PROGRAM BancoDeDados
VAR_INPUT
	InsertMarcha: InsertBD_Comandos;
	InsertParada: InsertBD_Comandos;
	ComandoSalvar:ARRAY[1..200] OF BOOL;
	bExecuteInsert		: BOOL; 
END_VAR
VAR
	Parte1Comandos	:STRING[100];
	Parte2Comandos	:STRING;
	Parte3Comandos	:STRING;
	RecordInsert	:FB_DBRecordInsert_EX;
	sCmdInsert		:T_MaxString;
	bInsertBusy		:BOOL;
	bInsertError	:BOOL;
	bInsertErrID	:UDINT;
	nRecords		:UDINT;
	
	Teste: BOOL;
END_VAR



//Código de erro 1142 - Usuário sem permissão para fazer o insert
//Código de erro 1146 - Tabela não encontrada
//Código de erro 1064 - Erro de sintaxe

//Pedaços do comando SQL para ficar melhor a montagem no uso delas
Parte1Comandos := 'INSERT INTO `comandos` (`comando`, `data_hora`, `usuario`, `serial_maquina`) VALUES (';
Parte2Comandos := CONCAT(', CURRENT_TIMESTAMP,$'', Main.NomeUsuario);
Parte3Comandos := CONCAT('$', $'', CONCAT(Main.SerialDaMaquina, '$')'));

RecordInsert(
	sNetID:= '127.0.0.1.1.1', //String containing the AMS network ID of the target device, at which the ADS command is directed.
	hDBID:= 1, // Indicates the ID of the database to be used.
	pCmdAddr:= ADR(sCmdInsert), //Pointer to the executing INSERT command
	cbCmdSize:= SIZEOF(sCmdInsert), //Indicates the length of the INSERT command.
	bExecute:= bExecuteInsert, 
	tTimeout:= T#5S, 
	bBusy=> bInsertBusy, 
	bError=> bInsertError, 
	nErrID=> bInsertErrID);
	

//----------------------- Comandos de funcionamento da máquina -----------------------//
{region "Comandos da máquina"}
//Marcha
bExecuteInsert := FALSE;
IF ComandoSalvar[1] THEN
	InsertMarcha(Insert:= TRUE, NomeComando:= 'MARCHA', InsertOut=> bExecuteInsert, Comando=> sCmdInsert);
	ComandoSalvar[1] := FALSE;
END_IF

//Parar
IF ComandoSalvar[2] THEN
	InsertParada(Insert:= TRUE, NomeComando:= 'PARADA', InsertOut=> bExecuteInsert, Comando=> sCmdInsert);
	ComandoSalvar[2] := FALSE;
END_IF

//Manual
IF ComandoSalvar[3] THEN
	InsertParada(Insert:= TRUE, NomeComando:= 'MAQ. EM MANUAL', InsertOut=> bExecuteInsert, Comando=> sCmdInsert);
	ComandoSalvar[3] := FALSE;
END_IF

//Auto
IF ComandoSalvar[4] THEN
	InsertParada(Insert:= TRUE, NomeComando:= 'MAQ. EM AUTOM.', InsertOut=> bExecuteInsert, Comando=> sCmdInsert);
	ComandoSalvar[4] := FALSE;
END_IF

//Fechar Ordem
IF ComandoSalvar[5] THEN
	InsertParada(Insert:= TRUE, NomeComando:= 'FECHAR ORDEM', InsertOut=> bExecuteInsert, Comando=> sCmdInsert);
	ComandoSalvar[5] := FALSE;
END_IF

//Aceitar lote
IF ComandoSalvar[6] THEN
	InsertParada(Insert:= TRUE, NomeComando:= 'ACEITAR LOTE', InsertOut=> bExecuteInsert, Comando=> sCmdInsert);
	ComandoSalvar[6] := FALSE;
END_IF

//Uma batelada
IF ComandoSalvar[7] THEN
	InsertParada(Insert:= TRUE, NomeComando:= 'UMA BATELADA', InsertOut=> bExecuteInsert, Comando=> sCmdInsert);
	ComandoSalvar[7] := FALSE;
END_IF

//Contínuo
IF ComandoSalvar[8] THEN
	InsertParada(Insert:= TRUE, NomeComando:= 'CONTÍNUO', InsertOut=> bExecuteInsert, Comando=> sCmdInsert);
	ComandoSalvar[8] := FALSE;
END_IF

//Pausa
IF ComandoSalvar[9] THEN
	InsertParada(Insert:= TRUE, NomeComando:= 'PAUSA', InsertOut=> bExecuteInsert, Comando=> sCmdInsert);
	ComandoSalvar[9] := FALSE;
END_IF
{endregion}


//----------------------- Acionamento manual das válvulas -----------------------//
{region "Válvulas Circuito 1"}
//------------------- Válvulas Circuito 1 -------------------//

//Circuito 1 Valvula 1 manual
IF ComandoSalvar[10] THEN
	InsertParada(Insert:= TRUE, NomeComando:= 'VALV. 1 CIRC. 1 MANUAL', InsertOut=> bExecuteInsert, Comando=> sCmdInsert);
	ComandoSalvar[10] := FALSE;
END_IF

//Circuito 1 Valvula 2 manual
IF ComandoSalvar[11] THEN
	InsertParada(Insert:= TRUE, NomeComando:= 'VALV. 2 CIRC. 1 MANUAL', InsertOut=> bExecuteInsert, Comando=> sCmdInsert);
	ComandoSalvar[11] := FALSE;
END_IF

//Circuito 1 Valvula 3 manual
IF ComandoSalvar[12] THEN
	InsertParada(Insert:= TRUE, NomeComando:= 'VALV. 3 CIRC. 1 MANUAL', InsertOut=> bExecuteInsert, Comando=> sCmdInsert);
	ComandoSalvar[12] := FALSE;
END_IF

//Circuito 1 Valvula 4 manual
IF ComandoSalvar[13] THEN
	InsertParada(Insert:= TRUE, NomeComando:= 'VALV. 4 CIRC. 1 MANUAL', InsertOut=> bExecuteInsert, Comando=> sCmdInsert);
	ComandoSalvar[13] := FALSE;
END_IF	  
{endregion}

{region "Válvulas Circuito 2"}
//------------------- Válvulas Circuito 2 -------------------//

//Circuito 2 Valvula 1 manual
IF ComandoSalvar[14] THEN
	InsertParada(Insert:= TRUE, NomeComando:= 'VALV. 1 CIRC. 2 MANUAL', InsertOut=> bExecuteInsert, Comando=> sCmdInsert);
	ComandoSalvar[14] := FALSE;
END_IF

//Circuito 2 Valvula 2 manual
IF ComandoSalvar[15] THEN
	InsertParada(Insert:= TRUE, NomeComando:= 'VALV. 2 CIRC. 2 MANUAL', InsertOut=> bExecuteInsert, Comando=> sCmdInsert);
	ComandoSalvar[15] := FALSE;
END_IF

//Circuito 2 Valvula 3 manual
IF ComandoSalvar[16] THEN
	InsertParada(Insert:= TRUE, NomeComando:= 'VALV. 3 CIRC. 2 MANUAL', InsertOut=> bExecuteInsert, Comando=> sCmdInsert);
	ComandoSalvar[16] := FALSE;
END_IF

//Circuito 2 Valvula 4 manual
IF ComandoSalvar[17] THEN
	InsertParada(Insert:= TRUE, NomeComando:= 'VALV. 4 CIRC. 2 MANUAL', InsertOut=> bExecuteInsert, Comando=> sCmdInsert);
	ComandoSalvar[17] := FALSE;
END_IF
{endregion}

{region "Válvulas Circuito 3"}
//------------------- Válvulas Circuito 3 -------------------//

//Circuito 3 Valvula 1 manual
IF ComandoSalvar[18] THEN
	InsertParada(Insert:= TRUE, NomeComando:= 'VALV. 1 CIRC. 3 MANUAL', InsertOut=> bExecuteInsert, Comando=> sCmdInsert);
	ComandoSalvar[18] := FALSE;
END_IF

//Circuito 3 Valvula 2 manual
IF ComandoSalvar[19] THEN
	InsertParada(Insert:= TRUE, NomeComando:= 'VALV. 2 CIRC. 3 MANUAL', InsertOut=> bExecuteInsert, Comando=> sCmdInsert);
	ComandoSalvar[19] := FALSE;
END_IF

//Circuito 3 Valvula 3 manual
IF ComandoSalvar[20] THEN
	InsertParada(Insert:= TRUE, NomeComando:= 'VALV. 3 CIRC. 3 MANUAL', InsertOut=> bExecuteInsert, Comando=> sCmdInsert);
	ComandoSalvar[20] := FALSE;
END_IF

//Circuito 3 Valvula 4 manual
IF ComandoSalvar[21] THEN
	InsertParada(Insert:= TRUE, NomeComando:= 'VALV. 4 CIRC. 3 MANUAL', InsertOut=> bExecuteInsert, Comando=> sCmdInsert);
	ComandoSalvar[21] := FALSE;
END_IF
{endregion}

{region "Válvulas Circuito 4"}
//------------------- Válvulas Circuito 4 -------------------//

//Circuito 4 Valvula 1 manual
IF ComandoSalvar[22] THEN
	InsertParada(Insert:= TRUE, NomeComando:= 'VALV. 1 CIRC. 4 MANUAL', InsertOut=> bExecuteInsert, Comando=> sCmdInsert);
	ComandoSalvar[22] := FALSE;
END_IF

//Circuito 4 Valvula 2 manual
IF ComandoSalvar[23] THEN
	InsertParada(Insert:= TRUE, NomeComando:= 'VALV. 2 CIRC. 4 MANUAL', InsertOut=> bExecuteInsert, Comando=> sCmdInsert);
	ComandoSalvar[23] := FALSE;
END_IF

//Circuito 4 Valvula 3 manual
IF ComandoSalvar[24] THEN
	InsertParada(Insert:= TRUE, NomeComando:= 'VALV. 3 CIRC. 4 MANUAL', InsertOut=> bExecuteInsert, Comando=> sCmdInsert);
	ComandoSalvar[24] := FALSE;
END_IF

//Circuito 4 Valvula 4 manual
IF ComandoSalvar[25] THEN
	InsertParada(Insert:= TRUE, NomeComando:= 'VALV. 4 CIRC. 4 MANUAL', InsertOut=> bExecuteInsert, Comando=> sCmdInsert);
	ComandoSalvar[25] := FALSE;
END_IF
{endregion}

{region "Válvulas Circuito 5"}
//------------------- Válvulas Circuito 5 -------------------//

//Circuito 5 Valvula 1 manual
IF ComandoSalvar[26] THEN
	InsertParada(Insert:= TRUE, NomeComando:= 'VALV. 1 CIRC. 5 MANUAL', InsertOut=> bExecuteInsert, Comando=> sCmdInsert);
	ComandoSalvar[26] := FALSE;
END_IF

//Circuito 5 Valvula 2 manual
IF ComandoSalvar[27] THEN
	InsertParada(Insert:= TRUE, NomeComando:= 'VALV. 2 CIRC. 5 MANUAL', InsertOut=> bExecuteInsert, Comando=> sCmdInsert);
	ComandoSalvar[27] := FALSE;
END_IF

//Circuito 5 Valvula 3 manual
IF ComandoSalvar[28] THEN
	InsertParada(Insert:= TRUE, NomeComando:= 'VALV. 3 CIRC. 5 MANUAL', InsertOut=> bExecuteInsert, Comando=> sCmdInsert);
	ComandoSalvar[28] := FALSE;
END_IF

//Circuito 5 Valvula 4 manual
IF ComandoSalvar[29] THEN
	InsertParada(Insert:= TRUE, NomeComando:= 'VALV. 4 CIRC. 5 MANUAL', InsertOut=> bExecuteInsert, Comando=> sCmdInsert);
	ComandoSalvar[29] := FALSE;
END_IF
{endregion}

{region "Válvulas Circuito 6"}
//------------------- Válvulas Circuito 6 -------------------//

//Circuito 6 Valvula 1 manual
IF ComandoSalvar[30] THEN
	InsertParada(Insert:= TRUE, NomeComando:= 'VALV. 1 CIRC. 6 MANUAL', InsertOut=> bExecuteInsert, Comando=> sCmdInsert);
	ComandoSalvar[30] := FALSE;
END_IF

//Circuito 6 Valvula 2 manual
IF ComandoSalvar[31] THEN
	InsertParada(Insert:= TRUE, NomeComando:= 'VALV. 2 CIRC. 6 MANUAL', InsertOut=> bExecuteInsert, Comando=> sCmdInsert);
	ComandoSalvar[31] := FALSE;
END_IF

//Circuito 6 Valvula 3 manual
IF ComandoSalvar[32] THEN
	InsertParada(Insert:= TRUE, NomeComando:= 'VALV. 3 CIRC. 6 MANUAL', InsertOut=> bExecuteInsert, Comando=> sCmdInsert);
	ComandoSalvar[32] := FALSE;
END_IF

//Circuito 6 Valvula 4 manual
IF ComandoSalvar[33] THEN
	InsertParada(Insert:= TRUE, NomeComando:= 'VALV. 4 CIRC. 6 MANUAL', InsertOut=> bExecuteInsert, Comando=> sCmdInsert);
	ComandoSalvar[33] := FALSE;
END_IF
{endregion}

{region "Válvulas Circuito 7"}
//------------------- Válvulas Circuito 7 -------------------//

//Circuito 7 Valvula 1 manual
IF ComandoSalvar[34] THEN
	InsertParada(Insert:= TRUE, NomeComando:= 'VALV. 1 CIRC. 7 MANUAL', InsertOut=> bExecuteInsert, Comando=> sCmdInsert);
	ComandoSalvar[34] := FALSE;
END_IF

//Circuito 7 Valvula 2 manual
IF ComandoSalvar[35] THEN
	InsertParada(Insert:= TRUE, NomeComando:= 'VALV. 2 CIRC. 7 MANUAL', InsertOut=> bExecuteInsert, Comando=> sCmdInsert);
	ComandoSalvar[35] := FALSE;
END_IF

//Circuito 7 Valvula 3 manual
IF ComandoSalvar[36] THEN
	InsertParada(Insert:= TRUE, NomeComando:= 'VALV. 3 CIRC. 7 MANUAL', InsertOut=> bExecuteInsert, Comando=> sCmdInsert);
	ComandoSalvar[36] := FALSE;
END_IF
	 
//Circuito 7 Valvula 4 manual
IF ComandoSalvar[37] THEN
	InsertParada(Insert:= TRUE, NomeComando:= 'VALV. 4 CIRC. 7 MANUAL', InsertOut=> bExecuteInsert, Comando=> sCmdInsert);
	ComandoSalvar[37] := FALSE;
END_IF
{endregion}

{region "Válvulas Circuito 8"}
//------------------- Válvulas Circuito 8 -------------------//

//Circuito 8 Valvula 1 manual
IF ComandoSalvar[38] THEN
	InsertParada(Insert:= TRUE, NomeComando:= 'VALV. 1 CIRC. 8 MANUAL', InsertOut=> bExecuteInsert, Comando=> sCmdInsert);
	ComandoSalvar[38] := FALSE;
END_IF

//Circuito 8 Valvula 2 manual
IF ComandoSalvar[39] THEN
	InsertParada(Insert:= TRUE, NomeComando:= 'VALV. 2 CIRC. 8 MANUAL', InsertOut=> bExecuteInsert, Comando=> sCmdInsert);
	ComandoSalvar[39] := FALSE;
END_IF

//Circuito 8 Valvula 3 manual
IF ComandoSalvar[40] THEN
	InsertParada(Insert:= TRUE, NomeComando:= 'VALV. 3 CIRC. 8 MANUAL', InsertOut=> bExecuteInsert, Comando=> sCmdInsert);
	ComandoSalvar[40] := FALSE;
END_IF

//Circuito 8 Valvula 4 manual
IF ComandoSalvar[41] THEN
	InsertParada(Insert:= TRUE, NomeComando:= 'VALV. 4 CIRC. 8 MANUAL', InsertOut=> bExecuteInsert, Comando=> sCmdInsert);
	ComandoSalvar[41] := FALSE;
END_IF
{endregion}
	 

{region "Válvulas Circuito 9"}
//------------------- Válvulas Circuito 9 -------------------//

//Circuito 9 Valvula 1 manual
IF ComandoSalvar[42] THEN
	InsertParada(Insert:= TRUE, NomeComando:= 'VALV. 1 CIRC. 9 MANUAL', InsertOut=> bExecuteInsert, Comando=> sCmdInsert);
	ComandoSalvar[42] := FALSE;
END_IF

//Circuito 9 Valvula 2 manual
IF ComandoSalvar[43] THEN
	InsertParada(Insert:= TRUE, NomeComando:= 'VALV. 2 CIRC. 9 MANUAL', InsertOut=> bExecuteInsert, Comando=> sCmdInsert);
	ComandoSalvar[43] := FALSE;
END_IF

//Circuito 9 Valvula 3 manual
IF ComandoSalvar[44] THEN
	InsertParada(Insert:= TRUE, NomeComando:= 'VALV. 3 CIRC. 9 MANUAL', InsertOut=> bExecuteInsert, Comando=> sCmdInsert);
	ComandoSalvar[44] := FALSE;
END_IF

//Circuito 9 Valvula 4 manual
IF ComandoSalvar[45] THEN
	InsertParada(Insert:= TRUE, NomeComando:= 'VALV. 4 CIRC. 9 MANUAL', InsertOut=> bExecuteInsert, Comando=> sCmdInsert);
	ComandoSalvar[45] := FALSE;
END_IF
{endregion}
	 

{region "Válvulas Circuito 10"}
//------------------- Válvulas Circuito 10 -------------------//

//Circuito 10 Valvula 1 manual
IF ComandoSalvar[46] THEN
	InsertParada(Insert:= TRUE, NomeComando:= 'VALV. 1 CIRC. 10 MANUAL', InsertOut=> bExecuteInsert, Comando=> sCmdInsert);
	ComandoSalvar[46] := FALSE;
END_IF

//Circuito 10 Valvula 2 manual
IF ComandoSalvar[47] THEN
	InsertParada(Insert:= TRUE, NomeComando:= 'VALV. 2 CIRC. 10 MANUAL', InsertOut=> bExecuteInsert, Comando=> sCmdInsert);
	ComandoSalvar[47] := FALSE;
END_IF

//Circuito 10 Valvula 3 manual
IF ComandoSalvar[48] THEN
	InsertParada(Insert:= TRUE, NomeComando:= 'VALV. 3 CIRC. 10 MANUAL', InsertOut=> bExecuteInsert, Comando=> sCmdInsert);
	ComandoSalvar[48] := FALSE;
END_IF

//Circuito 10 Valvula 4 manual
IF ComandoSalvar[49] THEN
	InsertParada(Insert:= TRUE, NomeComando:= 'VALV. 4 CIRC. 10 MANUAL', InsertOut=> bExecuteInsert, Comando=> sCmdInsert);
	ComandoSalvar[49] := FALSE;
END_IF
{endregion}
	 

{region "Válvulas Circuito 11"}
//------------------- Válvulas Circuito 11 -------------------//

//Circuito 11 Valvula 1 manual
IF ComandoSalvar[50] THEN
	InsertParada(Insert:= TRUE, NomeComando:= 'VALV. 1 CIRC. 11 MANUAL', InsertOut=> bExecuteInsert, Comando=> sCmdInsert);
	ComandoSalvar[50] := FALSE;
END_IF

//Circuito 11 Valvula 2 manual
IF ComandoSalvar[51] THEN
	InsertParada(Insert:= TRUE, NomeComando:= 'VALV. 2 CIRC. 11 MANUAL', InsertOut=> bExecuteInsert, Comando=> sCmdInsert);
	ComandoSalvar[51] := FALSE;
END_IF

//Circuito 11 Valvula 3 manual
IF ComandoSalvar[52] THEN
	InsertParada(Insert:= TRUE, NomeComando:= 'VALV. 3 CIRC. 11 MANUAL', InsertOut=> bExecuteInsert, Comando=> sCmdInsert);
	ComandoSalvar[52] := FALSE;
END_IF

//Circuito 11 Valvula 4 manual
IF ComandoSalvar[53] THEN
	InsertParada(Insert:= TRUE, NomeComando:= 'VALV. 4 CIRC. 11 MANUAL', InsertOut=> bExecuteInsert, Comando=> sCmdInsert);
	ComandoSalvar[53] := FALSE;
END_IF
{endregion}
	 

{region "Válvulas Circuito 12"}
//------------------- Válvulas Circuito 12 -------------------//

//Circuito 12 Valvula 1 manual
IF ComandoSalvar[54] THEN
	InsertParada(Insert:= TRUE, NomeComando:= 'VALV. 1 CIRC. 12 MANUAL', InsertOut=> bExecuteInsert, Comando=> sCmdInsert);
	ComandoSalvar[54] := FALSE;
END_IF

//Circuito 12 Valvula 2 manual
IF ComandoSalvar[55] THEN
	InsertParada(Insert:= TRUE, NomeComando:= 'VALV. 2 CIRC. 12 MANUAL', InsertOut=> bExecuteInsert, Comando=> sCmdInsert);
	ComandoSalvar[55] := FALSE;
END_IF

//Circuito 12 Valvula 3 manual
IF ComandoSalvar[56] THEN
	InsertParada(Insert:= TRUE, NomeComando:= 'VALV. 3 CIRC. 12 MANUAL', InsertOut=> bExecuteInsert, Comando=> sCmdInsert);
	ComandoSalvar[56] := FALSE;
END_IF

//Circuito 12 Valvula 4 manual
IF ComandoSalvar[57] THEN
	InsertParada(Insert:= TRUE, NomeComando:= 'VALV. 4 CIRC. 12 MANUAL', InsertOut=> bExecuteInsert, Comando=> sCmdInsert);
	ComandoSalvar[57] := FALSE;
END_IF
{endregion}


//-----------------------			Acionamento manual das válvulas de água			-----------------------//
{region "Válvulas de água"}
//Válvula de água limpa
IF ComandoSalvar[58] THEN
	InsertParada(Insert:= TRUE, NomeComando:= 'VALV. AGUA LIMPA MANUAL', InsertOut=> bExecuteInsert, Comando=> sCmdInsert);
	ComandoSalvar[58] := FALSE;
END_IF

//Válvula de água residual
IF ComandoSalvar[59] THEN
	InsertParada(Insert:= TRUE, NomeComando:= 'VALV. 4 AGUA RESID. MANUAL', InsertOut=> bExecuteInsert, Comando=> sCmdInsert);
	ComandoSalvar[59] := FALSE;
END_IF
{endregion}
	 

//-----------------------			Acionamento manual das bombas de dosagem		-----------------------//
{region "Bombas de dosagem"}
//Bomba da linha 1
IF ComandoSalvar[60] THEN
	InsertParada(Insert:= TRUE, NomeComando:= 'BOMBA DOSAD. 1 MANUAL', InsertOut=> bExecuteInsert, Comando=> sCmdInsert);
	ComandoSalvar[60] := FALSE;
END_IF	
//Bomba da linha 2 
IF ComandoSalvar[61] THEN
	InsertParada(Insert:= TRUE, NomeComando:= 'BOMBA DOSAD. 2 MANUAL', InsertOut=> bExecuteInsert, Comando=> sCmdInsert);
	ComandoSalvar[61] := FALSE;
END_IF	 
//Bomba da linha 3
IF ComandoSalvar[62] THEN
	InsertParada(Insert:= TRUE, NomeComando:= 'BOMBA DOSAD. 3 MANUAL', InsertOut=> bExecuteInsert, Comando=> sCmdInsert);
	ComandoSalvar[62] := FALSE;
END_IF	 
//Bomba da linha 4
IF ComandoSalvar[63] THEN
	InsertParada(Insert:= TRUE, NomeComando:= 'BOMBA DOSAD. 4 MANUAL', InsertOut=> bExecuteInsert, Comando=> sCmdInsert);
	ComandoSalvar[63] := FALSE;
END_IF	 
//Bomba da linha 5
IF ComandoSalvar[64] THEN
	InsertParada(Insert:= TRUE, NomeComando:= 'BOMBA DOSAD. 5 MANUAL', InsertOut=> bExecuteInsert, Comando=> sCmdInsert);
	ComandoSalvar[64] := FALSE;
END_IF	 
//Bomba da linha 6
IF ComandoSalvar[65] THEN
	InsertParada(Insert:= TRUE, NomeComando:= 'BOMBA DOSAD. 6 MANUAL', InsertOut=> bExecuteInsert, Comando=> sCmdInsert);
	ComandoSalvar[65] := FALSE;
END_IF	 
//Bomba da linha 7
IF ComandoSalvar[66] THEN
	InsertParada(Insert:= TRUE, NomeComando:= 'BOMBA DOSAD. 7 MANUAL', InsertOut=> bExecuteInsert, Comando=> sCmdInsert);
	ComandoSalvar[66] := FALSE;
END_IF	 
//Bomba da linha 8
IF ComandoSalvar[67] THEN
	InsertParada(Insert:= TRUE, NomeComando:= 'BOMBA DOSAD. 8 MANUAL', InsertOut=> bExecuteInsert, Comando=> sCmdInsert);
	ComandoSalvar[67] := FALSE;
END_IF	 
//Bomba da linha 9
IF ComandoSalvar[68] THEN
	InsertParada(Insert:= TRUE, NomeComando:= 'BOMBA DOSAD. 9 MANUAL', InsertOut=> bExecuteInsert, Comando=> sCmdInsert);
	ComandoSalvar[68] := FALSE;
END_IF	 
//Bomba da linha 10
IF ComandoSalvar[69] THEN
	InsertParada(Insert:= TRUE, NomeComando:= 'BOMBA DOSAD. 10 MANUAL', InsertOut=> bExecuteInsert, Comando=> sCmdInsert);
	ComandoSalvar[69] := FALSE;
END_IF	 
//Bomba da linha 11
IF ComandoSalvar[70] THEN
	InsertParada(Insert:= TRUE, NomeComando:= 'BOMBA DOSAD. 11 MANUAL', InsertOut=> bExecuteInsert, Comando=> sCmdInsert);
	ComandoSalvar[70] := FALSE;
END_IF	 
//Bomba da linha 12
IF ComandoSalvar[71] THEN
	InsertParada(Insert:= TRUE, NomeComando:= 'BOMBA DOSAD. 12 MANUAL', InsertOut=> bExecuteInsert, Comando=> sCmdInsert);
	ComandoSalvar[71] := FALSE;
END_IF
{endregion}

//-----------------------			Acionamento manual dos agitadores				-----------------------//
{region "Agitadores"}
//Agitador da linha 1
IF ComandoSalvar[72] THEN
	InsertParada(Insert:= TRUE, NomeComando:= 'AGITADOR 1 MANUAL', InsertOut=> bExecuteInsert, Comando=> sCmdInsert);
	ComandoSalvar[72] := FALSE;
END_IF
//Agitador da linha 2
IF ComandoSalvar[73] THEN
	InsertParada(Insert:= TRUE, NomeComando:= 'AGITADOR 2 MANUAL', InsertOut=> bExecuteInsert, Comando=> sCmdInsert);
	ComandoSalvar[73] := FALSE;
END_IF
//Agitador da linha 3
IF ComandoSalvar[74] THEN
	InsertParada(Insert:= TRUE, NomeComando:= 'AGITADOR 3 MANUAL', InsertOut=> bExecuteInsert, Comando=> sCmdInsert);
	ComandoSalvar[74] := FALSE;
END_IF
//Agitador da linha 4
IF ComandoSalvar[75] THEN
	InsertParada(Insert:= TRUE, NomeComando:= 'AGITADOR 4 MANUAL', InsertOut=> bExecuteInsert, Comando=> sCmdInsert);
	ComandoSalvar[75] := FALSE;
END_IF
//Agitador da linha 5
IF ComandoSalvar[76] THEN
	InsertParada(Insert:= TRUE, NomeComando:= 'AGITADOR 5 MANUAL', InsertOut=> bExecuteInsert, Comando=> sCmdInsert);
	ComandoSalvar[76] := FALSE;
END_IF
//Agitador da linha 6
IF ComandoSalvar[77] THEN
	InsertParada(Insert:= TRUE, NomeComando:= 'AGITADOR 6 MANUAL', InsertOut=> bExecuteInsert, Comando=> sCmdInsert);
	ComandoSalvar[77] := FALSE;
END_IF
//Agitador da linha 7
IF ComandoSalvar[78] THEN
	InsertParada(Insert:= TRUE, NomeComando:= 'AGITADOR 7 MANUAL', InsertOut=> bExecuteInsert, Comando=> sCmdInsert);
	ComandoSalvar[78] := FALSE;
END_IF
//Agitador da linha 8
IF ComandoSalvar[79] THEN
	InsertParada(Insert:= TRUE, NomeComando:= 'AGITADOR 8 MANUAL', InsertOut=> bExecuteInsert, Comando=> sCmdInsert);
	ComandoSalvar[79] := FALSE;
END_IF
//Agitador da linha 9
IF ComandoSalvar[80] THEN
	InsertParada(Insert:= TRUE, NomeComando:= 'AGITADOR 9 MANUAL', InsertOut=> bExecuteInsert, Comando=> sCmdInsert);
	ComandoSalvar[80] := FALSE;
END_IF
//Agitador da linha 10
IF ComandoSalvar[81] THEN
	InsertParada(Insert:= TRUE, NomeComando:= 'AGITADOR 10 MANUAL', InsertOut=> bExecuteInsert, Comando=> sCmdInsert);
	ComandoSalvar[81] := FALSE;
END_IF
//Agitador da linha 11
IF ComandoSalvar[82] THEN
	InsertParada(Insert:= TRUE, NomeComando:= 'AGITADOR 11 MANUAL', InsertOut=> bExecuteInsert, Comando=> sCmdInsert);
	ComandoSalvar[82] := FALSE;
END_IF
//Agitador da linha 12
IF ComandoSalvar[83] THEN
	InsertParada(Insert:= TRUE, NomeComando:= 'AGITADOR 12 MANUAL', InsertOut=> bExecuteInsert, Comando=> sCmdInsert);
	ComandoSalvar[83] := FALSE;
END_IF
{endregion}

//-----------------------			Inicia lavagem nas linhas						-----------------------//
{region "Inicio de lavagem"}
//Inicio da lavagem da linha 1
IF ComandoSalvar[84] THEN
	InsertParada(Insert:= TRUE, NomeComando:= 'INICIO LAV. L1', InsertOut=> bExecuteInsert, Comando=> sCmdInsert);
	ComandoSalvar[84] := FALSE;
END_IF	
//Inicio da lavagem da linha 2 
IF ComandoSalvar[85] THEN
	InsertParada(Insert:= TRUE, NomeComando:= 'INICIO LAV. L2', InsertOut=> bExecuteInsert, Comando=> sCmdInsert);
	ComandoSalvar[85] := FALSE;
END_IF
//Inicio da lavagem da linha 3
IF ComandoSalvar[86] THEN
	InsertParada(Insert:= TRUE, NomeComando:= 'INICIO LAV. L3', InsertOut=> bExecuteInsert, Comando=> sCmdInsert);
	ComandoSalvar[86] := FALSE;
END_IF	 
//Inicio da lavagem da linha 4
IF ComandoSalvar[87] THEN
	InsertParada(Insert:= TRUE, NomeComando:= 'INICIO LAV. L4', InsertOut=> bExecuteInsert, Comando=> sCmdInsert);
	ComandoSalvar[87] := FALSE;
END_IF	 
//Inicio da lavagem da linha 5
IF ComandoSalvar[88] THEN
	InsertParada(Insert:= TRUE, NomeComando:= 'INICIO LAV. L5', InsertOut=> bExecuteInsert, Comando=> sCmdInsert);
	ComandoSalvar[88] := FALSE;
END_IF	 
//Inicio da lavagem da linha 6
IF ComandoSalvar[89] THEN
	InsertParada(Insert:= TRUE, NomeComando:= 'INICIO LAV. L6', InsertOut=> bExecuteInsert, Comando=> sCmdInsert);
	ComandoSalvar[89] := FALSE;
END_IF	 
//Inicio da lavagem da linha 7
IF ComandoSalvar[90] THEN
	InsertParada(Insert:= TRUE, NomeComando:= 'INICIO LAV. L7', InsertOut=> bExecuteInsert, Comando=> sCmdInsert);
	ComandoSalvar[90] := FALSE;
END_IF	 
//Inicio da lavagem da linha 8
IF ComandoSalvar[91] THEN
	InsertParada(Insert:= TRUE, NomeComando:= 'INICIO LAV. L8', InsertOut=> bExecuteInsert, Comando=> sCmdInsert);
	ComandoSalvar[91] := FALSE;
END_IF
//Inicio da lavagem da linha 9
IF ComandoSalvar[92] THEN
	InsertParada(Insert:= TRUE, NomeComando:= 'INICIO LAV. L9', InsertOut=> bExecuteInsert, Comando=> sCmdInsert);
	ComandoSalvar[92] := FALSE;
END_IF 
//Inicio da lavagem da linha 10
IF ComandoSalvar[93] THEN
	InsertParada(Insert:= TRUE, NomeComando:= 'INICIO LAV. L10', InsertOut=> bExecuteInsert, Comando=> sCmdInsert);
	ComandoSalvar[93] := FALSE;
END_IF
//Inicio da lavagem da linha 11
IF ComandoSalvar[94] THEN
	InsertParada(Insert:= TRUE, NomeComando:= 'INICIO LAV. L11', InsertOut=> bExecuteInsert, Comando=> sCmdInsert);
	ComandoSalvar[94] := FALSE;
END_IF
//Inicio da lavagem da linha 12
IF ComandoSalvar[95] THEN
	InsertParada(Insert:= TRUE, NomeComando:= 'INICIO LAV. L12', InsertOut=> bExecuteInsert, Comando=> sCmdInsert);
	ComandoSalvar[95] := FALSE;
END_IF
{endregion}

//-----------------------			Para lavagem nas linhas							-----------------------//
{Region "Para a lavagem"}
//Parada da lavagem da linha 1
IF ComandoSalvar[96] THEN
	InsertParada(Insert:= TRUE, NomeComando:= 'PARA LAV. L1', InsertOut=> bExecuteInsert, Comando=> sCmdInsert);
	ComandoSalvar[96] := FALSE;
END_IF	
//Parada da lavagem da linha 2
IF ComandoSalvar[97] THEN
	InsertParada(Insert:= TRUE, NomeComando:= 'PARA LAV. L2', InsertOut=> bExecuteInsert, Comando=> sCmdInsert);
	ComandoSalvar[97] := FALSE;
END_IF	
//Parada da lavagem da linha 3
IF ComandoSalvar[98] THEN
	InsertParada(Insert:= TRUE, NomeComando:= 'PARA LAV. L3', InsertOut=> bExecuteInsert, Comando=> sCmdInsert);
	ComandoSalvar[98] := FALSE;
END_IF	
//Parada da lavagem da linha 4
IF ComandoSalvar[99] THEN
	InsertParada(Insert:= TRUE, NomeComando:= 'PARA LAV. L4', InsertOut=> bExecuteInsert, Comando=> sCmdInsert);
	ComandoSalvar[99] := FALSE;
END_IF	
//Parada da lavagem da linha 5
IF ComandoSalvar[100] THEN
	InsertParada(Insert:= TRUE, NomeComando:= 'PARA LAV. L5', InsertOut=> bExecuteInsert, Comando=> sCmdInsert);
	ComandoSalvar[100] := FALSE;
END_IF	
//Parada da lavagem da linha 6
IF ComandoSalvar[101] THEN
	InsertParada(Insert:= TRUE, NomeComando:= 'PARA LAV. L6', InsertOut=> bExecuteInsert, Comando=> sCmdInsert);
	ComandoSalvar[101] := FALSE;
END_IF	
//Parada da lavagem da linha 7
IF ComandoSalvar[102] THEN
	InsertParada(Insert:= TRUE, NomeComando:= 'PARA LAV. L7', InsertOut=> bExecuteInsert, Comando=> sCmdInsert);
	ComandoSalvar[102] := FALSE;
END_IF	
//Parada da lavagem da linha 8
IF ComandoSalvar[103] THEN
	InsertParada(Insert:= TRUE, NomeComando:= 'PARA LAV. L8', InsertOut=> bExecuteInsert, Comando=> sCmdInsert);
	ComandoSalvar[103] := FALSE;
END_IF	
//Parada da lavagem da linha 9
IF ComandoSalvar[104] THEN
	InsertParada(Insert:= TRUE, NomeComando:= 'PARA LAV. L9', InsertOut=> bExecuteInsert, Comando=> sCmdInsert);
	ComandoSalvar[104] := FALSE;
END_IF	
//Parada da lavagem da linha 10
IF ComandoSalvar[105] THEN
	InsertParada(Insert:= TRUE, NomeComando:= 'PARA LAV. L10', InsertOut=> bExecuteInsert, Comando=> sCmdInsert);
	ComandoSalvar[105] := FALSE;
END_IF	
//Parada da lavagem da linha 11
IF ComandoSalvar[106] THEN
	InsertParada(Insert:= TRUE, NomeComando:= 'PARA LAV. L11', InsertOut=> bExecuteInsert, Comando=> sCmdInsert);
	ComandoSalvar[106] := FALSE;
END_IF	
//Parada da lavagem da linha 12
IF ComandoSalvar[107] THEN
	InsertParada(Insert:= TRUE, NomeComando:= 'PARA LAV. L12', InsertOut=> bExecuteInsert, Comando=> sCmdInsert);
	ComandoSalvar[107] := FALSE;
END_IF	
{endregion}

//-----------------------			Acionamento manual dos elevadores				-----------------------//
{Region "Acionamento Elevadores"}
//Acionamento manual do elevador 1
IF ComandoSalvar[108] THEN
	InsertParada(Insert:= TRUE, NomeComando:= 'ACION. MANUAL ELEV1', InsertOut=> bExecuteInsert, Comando=> sCmdInsert);
	ComandoSalvar[108] := FALSE;
END_IF	
//Acionamento manual do elevador 2
IF ComandoSalvar[109] THEN
	InsertParada(Insert:= TRUE, NomeComando:= 'ACION. MANUAL ELEV2', InsertOut=> bExecuteInsert, Comando=> sCmdInsert);
	ComandoSalvar[109] := FALSE;
END_IF
//Acionamento manual do elevador 3
IF ComandoSalvar[110] THEN
	InsertParada(Insert:= TRUE, NomeComando:= 'ACION. MANUAL ELEV3', InsertOut=> bExecuteInsert, Comando=> sCmdInsert);
	ComandoSalvar[110] := FALSE;
END_IF
{endregion}
	 

//-----------------------			Descargas										-----------------------//
{Region "Descargas"}
//Caixa de recebimento
IF ComandoSalvar[111] THEN
	InsertParada(Insert:= TRUE, NomeComando:= 'ACION. MANUAL CX. RECEB.', InsertOut=> bExecuteInsert, Comando=> sCmdInsert);
	ComandoSalvar[111] := FALSE;
END_IF
//Caixa de 30Ton
IF ComandoSalvar[112] THEN
	InsertParada(Insert:= TRUE, NomeComando:= 'ACION. MANUAL CX. 30TON', InsertOut=> bExecuteInsert, Comando=> sCmdInsert);
	ComandoSalvar[112] := FALSE;
END_IF
//Caixa superior
IF ComandoSalvar[113] THEN
	InsertParada(Insert:= TRUE, NomeComando:= 'ACION. MANUAL CX. SUPERIOR', InsertOut=> bExecuteInsert, Comando=> sCmdInsert);
	ComandoSalvar[113] := FALSE;
END_IF
{endregion}
	 
	 

//-----------------------			Comandos das receitas							-----------------------//
{Region "Comandos das receitas"}
//Salvar
IF ComandoSalvar[114] THEN
	InsertParada(Insert:= TRUE, NomeComando:= 'SALVAR RECEITA', InsertOut=> bExecuteInsert, Comando=> sCmdInsert);
	ComandoSalvar[114] := FALSE;
END_IF
//Carregar
IF ComandoSalvar[115] THEN
	InsertParada(Insert:= TRUE, NomeComando:= 'CARREGAR RECEITA', InsertOut=> bExecuteInsert, Comando=> sCmdInsert);
	ComandoSalvar[115] := FALSE;
END_IF
//Excluir
IF ComandoSalvar[116] THEN
	InsertParada(Insert:= TRUE, NomeComando:= 'EXCLUIR RECEITA', InsertOut=> bExecuteInsert, Comando=> sCmdInsert);
	ComandoSalvar[116] := FALSE;
END_IF
{endregion}

//-----------------------			Confirmação dos alarmes							-----------------------//
{Region "Comandos da balança"}
//Confirma alarmes
IF ComandoSalvar[117] THEN
	InsertParada(Insert:= TRUE, NomeComando:= 'CONFIRMAR ALARMES', InsertOut=> bExecuteInsert, Comando=> sCmdInsert);
	ComandoSalvar[117] := FALSE;
END_IF

//-----------------------			Comandos da balança			-----------------------//
//Confirma alarmes
IF ComandoSalvar[117] THEN
	InsertParada(Insert:= TRUE, NomeComando:= 'CORTE GROSSO', InsertOut=> bExecuteInsert, Comando=> sCmdInsert);
	ComandoSalvar[117] := FALSE;
END_IF
//Confirma alarmes
IF ComandoSalvar[117] THEN
	InsertParada(Insert:= TRUE, NomeComando:= 'CORTE FINO', InsertOut=> bExecuteInsert, Comando=> sCmdInsert);
	ComandoSalvar[117] := FALSE;
END_IF
//Confirma alarmes
IF ComandoSalvar[117] THEN
	InsertParada(Insert:= TRUE, NomeComando:= 'PESO PADRÃO', InsertOut=> bExecuteInsert, Comando=> sCmdInsert);
	ComandoSalvar[117] := FALSE;
END_IF
//Confirma alarmes
IF ComandoSalvar[117] THEN
	InsertParada(Insert:= TRUE, NomeComando:= 'CONFIRMAR ALARMES', InsertOut=> bExecuteInsert, Comando=> sCmdInsert);
	ComandoSalvar[117] := FALSE;
END_IF
{endregion}

//-----------------------			Misturador							-----------------------//
{Region "Misturador"}
//Soprador
IF ComandoSalvar[118] THEN
	InsertParada(Insert:= TRUE, NomeComando:= 'SOPRADOR MANUAL', InsertOut=> bExecuteInsert, Comando=> sCmdInsert);
	ComandoSalvar[118] := FALSE;
END_IF
	//Prato
IF ComandoSalvar[119] THEN
	InsertParada(Insert:= TRUE, NomeComando:= 'PRATO MANUAL', InsertOut=> bExecuteInsert, Comando=> sCmdInsert);
	ComandoSalvar[119] := FALSE;
END_IF
//Aspersor
IF ComandoSalvar[120] THEN
	InsertParada(Insert:= TRUE, NomeComando:= 'ASPERSOR MANUAL', InsertOut=> bExecuteInsert, Comando=> sCmdInsert);
	ComandoSalvar[120] := FALSE;
END_IF
//Descarga
IF ComandoSalvar[121] THEN
	InsertParada(Insert:= TRUE, NomeComando:= 'DESCARGA TRAT. MANUAL', InsertOut=> bExecuteInsert, Comando=> sCmdInsert);
	ComandoSalvar[121] := FALSE;
END_IF
{endregion}

END_PROGRAM

(* stored: Version 1.1.0.1, ProductVersion 3.1.4024.14
   POU BancoDeDados: Id {1c2da0d4-ddc2-4df4-87ae-678610d1e3c0}, SpecialFunc None *)
